TEXTLIST TextList_Process
  0 = 'Selec proc' | FR: 'Procédé sélectionné :' | EN: 'Selected process:'
  1 = 'step' | FR: 'Etape en cours :' | EN: 'Step in progress:'
  2 = 'layer' | FR: 'Couche :' | EN: 'Layer:'
  3 = 'start' | FR: 'Marche\nProduction' | EN: 'Start\nProduction'
  4 = 'stop' | FR: 'Arrêt\nProduction' | EN: 'Stop\nProduction'
  5 = 'inter' | FR: 'Interruption\nProduction' | EN: 'Break\nProduction'
  6 = 'resume' | FR: 'Reprise\nProduction' | EN: 'Resume\nProduction'
  7 = 'process name' | FR: 'Nom procédé' | EN: 'Process name'
  8 = 'etape' | FR: 'Etape' | EN: 'Step'
  9 = 'type etape' | FR: 'Type étape' | EN: 'Step type'
  10 = 'tps effluvage' | FR: 'Durée effluvage' | EN: 'Glow disch. time'
  11 = 'couche' | FR: 'Couche' | EN: 'Layer'
  12 = 'détails' | FR: 'Détails' | EN: 'Details'
  13 = 'boucle' | FR: 'Boucle' | EN: 'Loop'
  14 = 'first' | FR: 'Départ' | EN: 'First'
  15 = 'fin' | FR: 'Fin' | EN: 'Last'
  16 = 'seg' | FR: 'Segment' | EN: 'Segment'
  17 = 'tps seg' | FR: 'Temps segment' | EN: 'Segment time'
  18 = 'tps couche' | FR: 'Temps couche' | EN: 'Layer time'
  19 = 'next layer' | FR: 'Couche suivante' | EN: 'Next layer'
  20 = 'break' | FR: 'Interruption' | EN: 'Break'
  21 = 'resume' | FR: 'Reprise' | EN: 'Resume'
  22 = 'arrêt' | FR: 'Arrêt procédé' | EN: 'Process stop'
  23 = 'next step' | FR: 'Etape suivante' | EN: 'Next step'
  24 = 'Temps purge' | FR: 'Temps purge' | EN: 'Purge time'
  25 = 'Temps etching' | FR: 'Temps décapage' | EN: 'Etching time'
  26 = 'Rechargement' | FR: 'Rechargement' | EN: 'Reload'
   = ''
END_TEXTLIST

(* stored: Version 1.1.0.1, ProductVersion 3.1.4024.10
   TextList TextList_Process: Id {9d08fc89-6a7f-49bf-b64a-7b3df3733506} *)
